FUNCTION_BLOCK FB_MassFlowMonitor
VAR_IN_OUT
	fbSensors : ARRAY[1..GVL.massFlowSensorCount] OF ST_MassFlowSensor;
END_VAR

VAR
	fbScale : ARRAY[1..GVL.massFlowSensorCount] OF FB_ScaleAnalog;
	i : INT;
END_VAR

FOR i := 1 TO GVL.massFlowSensorCount DO
	fbScale[i](
		fbRawValue := fbSensors[i].RawValue,
		fbInputMin := fbSensors[i].InputMin,
		fbInputMax := fbSensors[i].InputMax,
		fbOutputMin := fbSensors[i].OutputMin,
		fbOutputMax := fbSensors[i].OutputMax,
		fbScaledValue => fbSensors[i].ScaledValue,
		fbRangeError => fbSensors[i].RangeError);
END_FOR

END_FUNCTION_BLOCK

(* stored: Version 1.1.0.1
   POU FB_MassFlowMonitor: Id {e5f6a7b8-9c0d-1e2f-3a4b-5c6d7e8f9a0b}, SpecialFunc None *)
